FUNCTION_BLOCK PUBLIC PAEScaleTotalizing EXTENDS PAEScaleGravimetric IMPLEMENTS IPAScaleTotalizing
VAR_INPUT
END_VAR
VAR_OUTPUT
END_VAR
VAR
	_IsFlow : BOOL;
	_IsPresignal : BOOL;
	_TotalActualWeight : LREAL;
	_TotalDesiredWeight : LREAL;
END_VAR

METHOD FB_postinit
VAR_INPUT
	root : IACVariobatch;
END_VAR
SUPER^.FB_postinit(root);
root.OnPropertyChangedLReal(THIS^, 86, _TotalDesiredWeight);
root.OnPropertyChangedLReal(THIS^, 87, _TotalActualWeight);
root.OnPropertyChangedBool(THIS^, 88, _IsPresignal);
root.OnPropertyChangedBool(THIS^, 89, _IsFlow);
END_METHOD

METHOD PUBLIC InvokeSetterBool
VAR_INPUT
	PropertyID : INT;
	PropertyValue : BOOL;
END_VAR
SUPER^.InvokeSetterBool(PropertyID, PropertyValue);
CASE PropertyID OF
	88:
		IsPresignal := PropertyValue;
	89:
		IsFlow := PropertyValue;
END_CASE
END_METHOD

METHOD PUBLIC InvokeSetterLReal
VAR_INPUT
	PropertyID : INT;
	PropertyValue : LREAL;
END_VAR
SUPER^.InvokeSetterLReal(PropertyID, PropertyValue);
CASE PropertyID OF
	86:
		TotalDesiredWeight := PropertyValue;
	87:
		TotalActualWeight := PropertyValue;
END_CASE
END_METHOD

{attribute 'monitoring' := 'call'}
//{attribute 'TcRpcEnable'}
PROPERTY PUBLIC IsFlow : BOOL
GET // PUBLIC
IsFlow := _IsFlow;
END_GET
SET // PUBLIC
_IsFlow := IsFlow;
Root.OnPropertyChangedBool(THIS^, 89, _IsFlow);
END_SET
END_PROPERTY

{attribute 'monitoring' := 'call'}
//{attribute 'TcRpcEnable'}
PROPERTY PUBLIC IsPresignal : BOOL
GET // PUBLIC
IsPresignal := _IsPresignal;
END_GET
SET // PUBLIC
_IsPresignal := IsPresignal;
Root.OnPropertyChangedBool(THIS^, 88, _IsPresignal);
END_SET
END_PROPERTY

METHOD OnInitMemory
VAR_INPUT
	root : IACVariobatch;
END_VAR
RegisterProperty(root, 86, GCL.cSizeLREAL); //TotalDesiredWeight
RegisterProperty(root, 87, GCL.cSizeLREAL); //TotalActualWeight
RegisterProperty(root, 88, GCL.cSizeBYTE); //IsPresignal
RegisterProperty(root, 89, GCL.cSizeBYTE); //IsFlow
SUPER^.OnInitMemory(root);
END_METHOD

{attribute 'monitoring' := 'call'}
//{attribute 'TcRpcEnable'}
PROPERTY PUBLIC TotalActualWeight : LREAL
GET // PUBLIC
TotalActualWeight := _TotalActualWeight;
END_GET
SET // PUBLIC
_TotalActualWeight := TotalActualWeight;
Root.OnPropertyChangedLReal(THIS^, 87, _TotalActualWeight);
END_SET
END_PROPERTY

{attribute 'monitoring' := 'call'}
//{attribute 'TcRpcEnable'}
PROPERTY PUBLIC TotalDesiredWeight : LREAL
GET // PUBLIC
TotalDesiredWeight := _TotalDesiredWeight;
END_GET
SET // PUBLIC
_TotalDesiredWeight := TotalDesiredWeight;
Root.OnPropertyChangedLReal(THIS^, 86, _TotalDesiredWeight);
END_SET
END_PROPERTY

END_FUNCTION_BLOCK

(* stored: Version 1.1.0.1, ProductVersion 3.1.4024.6
   POU PAEScaleTotalizing: Id {a9ca8691-6ed6-48b1-98f6-5baa3f5d4144}, SpecialFunc None
   Method FB_postinit: Id {c1e1d5ec-d137-469f-beee-ca90cf47ac68}
   Method InvokeSetterBool: Id {6c71a670-db73-43e1-a473-ec3e0e294366}
   Method InvokeSetterLReal: Id {82aac350-8ba4-468f-8abb-1e9f55edcaca}
   Property IsFlow: Id {5171db51-d421-44ad-9266-ac7b8380d43c}
   Get Get: Id {5ac95594-0695-4a0b-af47-6f453740fff7}
   Set Set: Id {f5f2c0bb-bd1e-4836-820a-fde6b3e29893}
   Property IsPresignal: Id {087e34b6-7f2c-4f3c-b484-1e92535cf8d2}
   Get Get: Id {0fed6fbe-2f1f-41fa-8e23-02f885514806}
   Set Set: Id {1da5fb6c-bb72-4833-bac9-7043683991e6}
   Method OnInitMemory: Id {97cbbab0-e2b4-4cdc-9783-1918016ffebf}
   Property TotalActualWeight: Id {6ae8eb58-1efd-4c2a-b16f-c707d2eeb87d}
   Get Get: Id {fd1c32e4-fca7-41b9-995b-b21cd9860cb8}
   Set Set: Id {93e3ed51-d8db-4d53-bc44-ee63ddada043}
   Property TotalDesiredWeight: Id {bed5e69d-1480-4c9b-acb5-eea6798acba1}
   Get Get: Id {de1ee27c-0bb9-463d-83d4-248242583844}
   Set Set: Id {1c5e0f7d-2194-4c84-b082-960b16e0cfbb} *)
